                       #T.TunnelAck.IP_Header.HeaderSize := 16#06;
                       #T.TunnelAck.IP_Header.ProtokollVersion := 16#10;
                       #T.TunnelAck.IP_Header.ServiceType := 16#0421;
                       #T.TunnelAck.IP_Header.TotalLaenge := 16#000A;

                       #T.TunnelAck.IP_Body.Laenge := 16#04;
                       #T.TunnelAck.IP_Body.ChannelID := #KNX.ChannelID;
                       #T.TunnelAck.IP_Body.SequenzCount := #KNX.SeqNrEmpf;
                       //#KNX.SeqNr := #T.Tunnel.Conn_Header.SequenzeCount;
                       #T.TunnelAck.IP_Body.Status := 16#0;

                       #POS := 0;
                       #fehler := Serialize(SRC_VARIABLE := #T.TunnelAck, DEST_ARRAY => #SendData, POS := #POS);

                       #SendeLaenge := #POS;
                       #Senden := true;

                   5: //Tunneltelegramm senden!
                       #T.Tunnel.IP_Header.HeaderSize := 16#06;
                       #T.Tunnel.IP_Header.ProtokollVersion := 16#10;
                       #T.Tunnel.IP_Header.ServiceType := 16#420;
                       #T.Tunnel.IP_Header.TotalLaenge := #KNX_Dat.Send_Dat.Laenge+20; //16#15;

                       #T.Tunnel.Conn_Header.Laenge := 04;
                       #T.Tunnel.Conn_Header.ChannelID := #KNX.ChannelID;
                       #T.Tunnel.Conn_Header.SequenzeCount := #KNX.SeqNrSenden;
                       #T.Tunnel.Conn_Header.Reserve := 16#00;

                       #T.Tunnel.Cemi.MessageCode := 16#11;
                       #T.Tunnel.Cemi.AdditionalLaenge := 16#00;
                       #T.Tunnel.Cemi.Kontrollbyte1 := 16#bC;
                       #T.Tunnel.Cemi.Kontrollbyte2 := 16#E0;
                       #T.Tunnel.Cemi.SourceAddr := 16#0000;
                       //#T.Tunnel.Cemi.DestinationAddr := 16#0506;
                       //#T.Tunnel.NPDU.Laenge := 16#01;
                       //#T.Tunnel.NPDU.NPDU_ABCI := 16#00;
                       //IF "Allg".EinAus THEN
                       //    #T.Tunnel.NPDU.Daten[1] := 16#81;
                       //ELSE
                       //    #T.Tunnel.NPDU.Daten[1] := 16#80;
                       //END_IF;

                #T.Tunnel.Cemi.DestinationAddr := #KNX_Dat.Send_Dat.GruppenAddr;
                #T.Tunnel.NPDU.Laenge := #KNX_Dat.Send_Dat.Laenge;
                #T.Tunnel.NPDU.NPDU_ABCI := #KNX_Dat.Send_Dat.NPDU_ABCI;
                #T.Tunnel.NPDU.Daten := #KNX_Dat.Send_Dat.Daten;
                       #POS := 0;
                       #fehler := Serialize(SRC_VARIABLE := #T.Tunnel, DEST_ARRAY => #SendData, POS := #POS);

                       #SendeLaenge := #KNX_Dat.Send_Dat.Laenge+20;
                       #Senden := true;
             6: //Tunnel-Abbau-Telegramm senden
                       #T.AnfTunnelState.IP_Header.HeaderSize := 16#06;
                       #T.AnfTunnelState.IP_Header.ProtokollVersion := 16#10;
                       #T.AnfTunnelState.IP_Header.ServiceType := 16#0209;
                       #T.AnfTunnelState.IP_Header.TotalLaenge := 16#0010;

                       #T.AnfTunnelState.IP_Body.CummunicationChannel := #KNX.ChannelID;
                       #T.AnfTunnelState.IP_Body.Reserve := 16#00;
                       #T.AnfTunnelState.IP_Body.Control_EndPoint.Laenge := 16#08;
                       #T.AnfTunnelState.IP_Body.Control_EndPoint.ProtocolCode := 16#01;
                       #T.AnfTunnelState.IP_Body.Control_EndPoint.IP1 := #EigeneIP[1];
                       #T.AnfTunnelState.IP_Body.Control_EndPoint.IP2 := #EigeneIP[2];
                       #T.AnfTunnelState.IP_Body.Control_EndPoint.IP3 := #EigeneIP[3];
                       #T.AnfTunnelState.IP_Body.Control_EndPoint.IP4 := #EigeneIP[4];
                       #T.AnfTunnelState.IP_Body.Control_EndPoint."Port" := #Port_Lokal;
                       #POS := 0;
                       #fehler := Serialize(SRC_VARIABLE := #T.AnfTunnelState, DEST_ARRAY => #SendData, POS := #POS);

                       #SendeLaenge := #POS;
                       #Senden := true;
           END_CASE;

   //Daten senden!
   #USEND(REQ := #Senden ,
                ID := #ConnID,
                LEN := DINT_TO_UDINT(#SendeLaenge),
                DATA := #SendData,
                ADDR := #KNX_Endpunkt);
   IF #USEND.ERROR THEN
       #Senden := false;
       #STATUS_USEND := #USEND.STATUS;
       #SendeAnf := 0;
   END_IF;
   IF  #USEND.DONE THEN
       #SendeAnf := 0;
       #Senden := false;
       #STATUS_USEND := 0;
       #KNXInfo.SendeTicks := #KNXInfo.SendeTicks + 1;
   END_IF;

   //Bausteinausgaben
   #Status := #State;
   #OK := #State >= 100 AND #State < 250;
   IF #IEC_Timer_TimeOut.Q THEN
       #HMTimeOut := true;
   END_IF;
   IF #URCV.NDR THEN
       #HMTimeOut := false;
   END_IF;
   #TimeOut := #HMTimeOut;
END_FUNCTION_BLOCK

FUNCTION_BLOCK "knx-KO"   // FB15, FBD
{ S7_Optimized_Access := 'TRUE' }
VERSION : 0.1
   VAR_IN_OUT
      Wert : Variant;   // Zu sendender / Empfangender Wert!
      KNX_KO : "KNX_KO";
      KNX_Dat : "KNX_Data_Exchange";
   END_VAR
   VAR
      "knx-SendByChange_Instance" : "knx-SendByChange";
      "knx-rxBus-GroupValueRead_Instance" : "knx-rxBus-GroupValueRead";
      "knx-txBus-GroupValueRead_Instance" : "knx-txBus-GroupValueRead";
      "knx-sendenEmpfangen_Instance" : "knx-sendenEmpfangen";
      fl_counterSend : Bool;
   END_VAR
   VAR_TEMP   // added for the SCL form of the ladder/FBD networks
      _w1 : Bool;
      _w2 : Bool;
   END_VAR
BEGIN

REGION Network 1 (SCL): INFO
   (*

   Sammelbaustein der das KO (Kommunikationsobjekt) zwischen SPS und Bus organisiert


   17.10.2021 van
   Auswertung des #KNX_KO.para.aktiv Bits

   04.10.2021 van
   Baustein erstellt

   *)
END_REGION

REGION Network 2: Aktiv
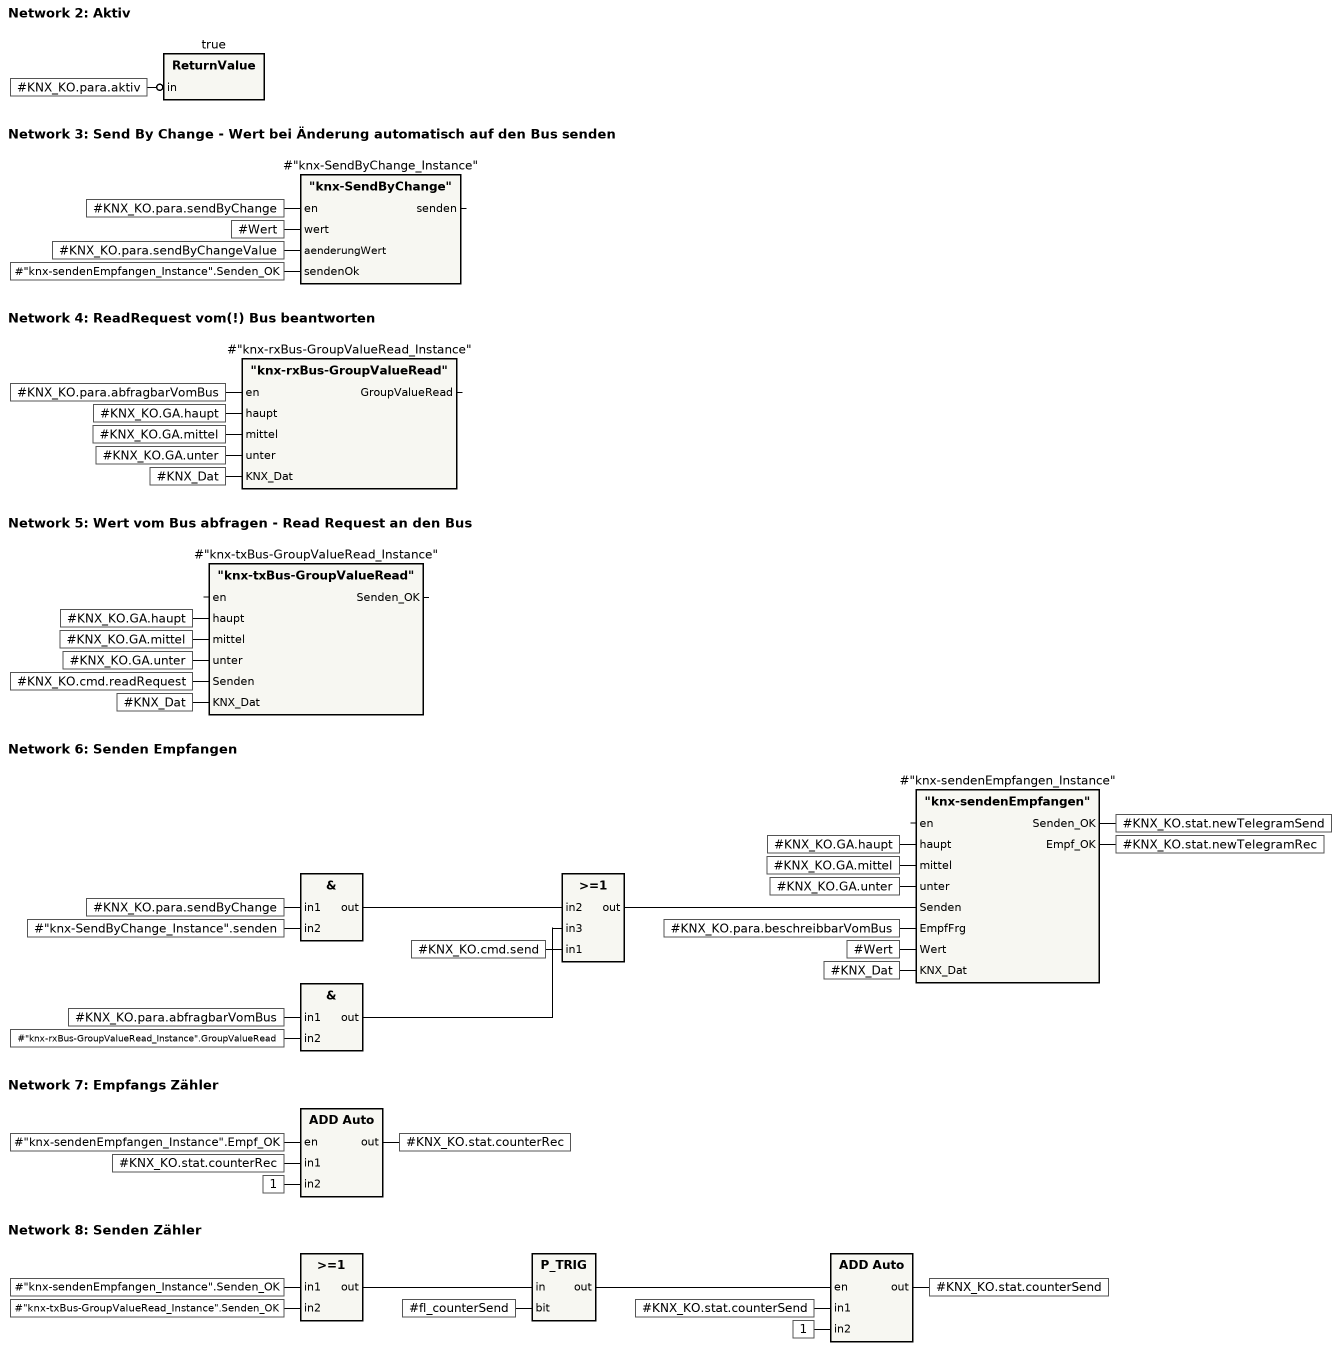
   IF NOT #KNX_KO.para.aktiv THEN
       ENO := true;
       RETURN;
   END_IF;
END_REGION

REGION Network 3: Send By Change - Wert bei Änderung automatisch auf den Bus senden
   IF #KNX_KO.para.sendByChange THEN
       #"knx-SendByChange_Instance"(wert := #Wert,   // "knx-SendByChange"
                               aenderungWert := #KNX_KO.para.sendByChangeValue,
                               sendenOk := #"knx-sendenEmpfangen_Instance".Senden_OK);
   END_IF;
END_REGION

REGION Network 4: ReadRequest vom(!) Bus beantworten
   IF #KNX_KO.para.abfragbarVomBus THEN
       #"knx-rxBus-GroupValueRead_Instance"(haupt := #KNX_KO.GA.haupt,   // "knx-rxBus-GroupValueRead"
                               mittel := #KNX_KO.GA.mittel,
                               unter := #KNX_KO.GA.unter,
                               KNX_Dat := #KNX_Dat);
   END_IF;
END_REGION

REGION Network 5: Wert vom Bus abfragen - Read Request an den Bus
   #"knx-txBus-GroupValueRead_Instance"(haupt := #KNX_KO.GA.haupt,   // "knx-txBus-GroupValueRead"
                           mittel := #KNX_KO.GA.mittel,
                           unter := #KNX_KO.GA.unter,
                           Senden := #KNX_KO.cmd.readRequest,
                           KNX_Dat := #KNX_Dat);
END_REGION

REGION Network 6: Senden Empfangen
   #"knx-sendenEmpfangen_Instance"(haupt := #KNX_KO.GA.haupt,   // "knx-sendenEmpfangen"
                           mittel := #KNX_KO.GA.mittel,
                           unter := #KNX_KO.GA.unter,
                           Senden := (#KNX_KO.para.sendByChange AND #"knx-SendByChange_Instance".senden) OR (#KNX_KO.para.abfragbarVomBus AND #"knx-rxBus-GroupValueRead_Instance".GroupValueRead) OR #KNX_KO.cmd.send,
                           EmpfFrg := #KNX_KO.para.beschreibbarVomBus,
                           Wert := #Wert,
                           KNX_Dat := #KNX_Dat,
                           Senden_OK => #KNX_KO.stat.newTelegramSend,
                           Empf_OK => #KNX_KO.stat.newTelegramRec);
END_REGION

REGION Network 7: Empfangs Zähler
   IF #"knx-sendenEmpfangen_Instance".Empf_OK THEN
       #KNX_KO.stat.counterRec := #KNX_KO.stat.counterRec + 1;
   END_IF;
END_REGION

REGION Network 8: Senden Zähler
   #_w1 := #"knx-sendenEmpfangen_Instance".Senden_OK OR #"knx-txBus-GroupValueRead_Instance".Senden_OK;
   #_w2 := #_w1 AND NOT #fl_counterSend;   // rising edge
   #fl_counterSend := #_w1;
   IF #_w2 THEN #KNX_KO.stat.counterSend := #KNX_KO.stat.counterSend + 1; END_IF;
END_REGION
END_FUNCTION_BLOCK

FUNCTION "knx-GAword-to-GAnr" : "KNX_GA_Nr"   // FC1, SCL
{ S7_Optimized_Access := 'TRUE' }
VERSION : 0.1
   VAR_INPUT
      GruppenAddr : Word;
   END_VAR
BEGIN

   (*

   Wandelt eine Dreistufige KNX GA (Word) in eine ihre Bestandteile (Haupt-, Mittel-, Untergruppe) auf 

   INFOS:

   https://support.knx.org/hc/de/articles/115003188109-Gruppenadressen

   3-Ebenen-Darstellung“ = Hauptgruppe/Mittelgruppe/Untergruppe

   Hauptgruppe = D7+D6+D5+D4+D3 des ersten Oktetts (hohe Adresse)
   Mittelgruppe = D2+D1+D0 des ersten Oktetts (hohe Adresse)
   Untergruppe = das gesamte zweite Oktett (niedrige Adresse)
   Bereiche: Hauptgruppe = 0..31, Mittelgruppe = 0..7, Untergruppe = 0..255

   Quelle:
   https://www.sps-forum.de/gebaeudeautomatisierung/93641-knx-kommunkation-ueber-knxnet-ip-mit-siemens-s7-1500-s7-1200-tia-portal-post704269.html#post704269

   *)



   #"knx-GAword-to-GAnr".haupt := SHR(IN := (#GruppenAddr AND 16#F800), N := 11);
   #"knx-GAword-to-GAnr".mittel := SHR(IN := (#GruppenAddr AND 16#700), N := 8);
   #"knx-GAword-to-GAnr".unter := #GruppenAddr AND 16#FF;
END_FUNCTION

FUNCTION "knx-GAnr-to-GAword" : Word   // FC2, SCL
{ S7_Optimized_Access := 'TRUE' }
VERSION : 0.1
   VAR_INPUT
      haupt : UInt;   // Hauptgruppe = 0..31
      mittel : UInt;   // Mittelgruppe = 0..7
      unter : UInt;   // Untergruppe = 0..255
   END_VAR
   VAR_TEMP
      GruppenAddr : Word;
   END_VAR
BEGIN

   (*

   Erstellt eine Dreistufige KNX GA (Word) aus den Bestandteilen (Haupt-, Mittel-, Untergruppe)

   Quelle:
   Aus "KNX_GruppeAddr" entnommen

   *)


   //Gruppenadresse zu einem Wort zusammenbauen!
   #GruppenAddr := SHL(IN := #haupt, N := 11);
   #GruppenAddr := #GruppenAddr OR SHL(IN := #mittel, N := 8);
   #GruppenAddr := #GruppenAddr OR #unter;


   #"knx-GAnr-to-GAword" := #GruppenAddr;
END_FUNCTION

FUNCTION "knx-real-to-DPT9" : Word   // FC3, SCL
{ S7_Optimized_Access := 'TRUE' }
VERSION : 0.1
   VAR_INPUT
      inReal : Real;
   END_VAR
   VAR_TEMP
      tmpExp : Int;
      tmpDIntValIn : DInt;
      tmp_dInt : DInt;
      tmpOut : Int;
   END_VAR
BEGIN

   (*

   Wandelt eine Real Zahl in den DPT9.xxx (2 Byte Gleitkommawert)

   Quelle:
   https://www.sps-forum.de/threads/knx-kommunkation-%C3%BCber-knxnet-ip-mit-siemens-s7-1500-s7-1200-tia-portal.93641/post-804342

   Weitere Infos:
   03_07_02 Datapoint Types v01.08.02 AS.pdf
   3.10 Datapoint Types “2-Octet Float Value”

   Range: [-671 088,64 … 670 760,96]


   03.10.2021 van
   Baustein erstellt anhand des Code von Oberchefe

   *)

   #tmpExp := 0;    (*    Exponent initialisieren    *)

   #tmpDIntValIn := REAL_TO_DINT(#inReal * 100.0);

   IF #tmpDIntValIn > 2047  THEN   // OR #tmpDIntValIn < -2048

       WHILE #tmpDIntValIn / (2**#tmpExp) > 2047 DO     //EXPT(2, #tmpExp)
           #tmpExp := #tmpExp + 1;
       END_WHILE;

   ELSIF #tmpDIntValIn < -2048 THEN

       WHILE #tmpDIntValIn / (2**#tmpExp) < -2048 DO    // EXPT(2, #tmpExp)
           #tmpExp := #tmpExp + 1;
       END_WHILE;

   ELSE            (*    Kein Exponent erforderlich    *)

       ;

   END_IF;


   #tmp_dInt := #tmpDIntValIn / REAL_TO_DINT((2**(#tmpExp)));         (*    Mantisse roh   *)  //(EXPT(2, INT_TO_WORD(#tmpExp))

   #tmp_dInt := WORD_TO_DINT(DINT_TO_WORD(#tmp_dInt) AND 16#7FF);
   #tmpOut := SHL(IN := #tmpExp, N:=11);                (*    Exponent positionieren        *)


   IF #tmpDIntValIn < 0 THEN                    (*    negativ?    -> Vorzeichen setzen    *)
       #tmpOut := #tmpOut OR 16#8000;
   END_IF;


   #"knx-real-to-DPT9":= #tmpOut OR DINT_TO_WORD(#tmp_dInt);
END_FUNCTION

FUNCTION "knx-DPT9-to-real" : Real   // FC4, SCL
{ S7_Optimized_Access := 'TRUE' }
VERSION : 0.1
   VAR_INPUT
      inWord : Word;
   END_VAR
   VAR_TEMP
      tmp_Word1 : Word;
      tmp_M : DWord;
      tmp_Dword : DWord;
      tmp_e2 : UDInt;
      tmp_Real : Real;
      tmp_Int : Int;
      tmpInt_M : Int;
      tmpInt_E : Int;
      tmpReal_M : Real;
      tmpReal_E : Real;
      tmpReal : Real;
   END_VAR
BEGIN
   (*

   Wandelt ein DPT9.xxx (2 Byte Gleitkommawert) in einen Real

   Weitere Infos:
   03_07_02 Datapoint Types v01.08.02 AS.pdf
   3.10 Datapoint Types “2-Octet Float Value”

   03.10.2021 van
   Baustein erstellt

   *)



   //Ergebnis = (0,01 * M)*2^E   //Siehe PDF 03_07_02 Kap. 3.10)
   // E = [0 … 15]
   // M = [-2 048 … 2 047], two’s complement notation

   (*

   76543210 76543210
   MEEEEMMM MMMMMMMM

   *)

   #tmp_Word1:= #inWord;

   // Mantisse
   #tmpInt_M := WORD_TO_INT(#tmp_Word1 & 16#07ff);
   #tmpReal_M := INT_TO_REAL(#tmpInt_M);

   //Negative Mantisse anpassen
   //Das muss noch irgendwie besser gehen ...
   IF #tmp_Word1.%X15 THEN
       #tmpReal_M := (#tmpReal_M*-1.0) + 2048.0;
   END_IF;


   // Exponent
   // #tmp_Dword := #tmp_Word1 & 16#7800;  //Exponent
   // #tmp_e2 := SHR(IN := #tmp_Dword, N := 11);

   #tmp_e2 := SHR(IN := SHL(IN := #tmp_Word1, N := 1), N := 12);

   #tmpInt_E := UDINT_TO_INT(#tmp_e2);
   #tmpReal_E := INT_TO_REAL(#tmpInt_E);


   // FloatValue = (0,01 * M)*2^E 
   #tmpReal := (0.01 * #tmpReal_M) * (2**#tmpReal_E);


   //Vorzeichen
   IF #tmp_Word1.%X15 THEN
       #tmpReal := (#tmpReal * -1.0) ;
   END_IF;


   #"knx-DPT9-to-real" := #tmpReal;
END_FUNCTION

FUNCTION "knx-DPT3-to-plc" : "KNX_DPT3"   // FC14, SCL
{ S7_Optimized_Access := 'TRUE' }
VERSION : 0.1
   VAR_INPUT
      data : Byte;   // RAW DPT3 Daten
   END_VAR
   VAR_TEMP
      tmpStepCode : USInt;
   END_VAR
   // Ret_Val : Aufbereitete DPT3 Daten
BEGIN
   (*

   knx-DPT3-to-plc

   Wandelt den DPT3 Wert vom KNX Bus in einen PLC "KNX_DPT3" Wert

   DPT 3   4 Bit   0..15     
   3.yyy = boolesch + vorzeichenloser 3-Bit-Wert, z. B. Auf-/Abdimmen  

   \The KNX Standard v2.1\The KNX Standard v2.1\03 Volume 3 System Specifications\
   03_07_02 Datapoint Types v01.08.02 AS.pdf
   3.3 Datapoint Types B1U3 


   20.02.2024 van
   Baustein erstellt

   *)

   (*** StepCode ***

   StepCode The amount of intervals into which the 
   range of 0 % … 100 % is subdivided, or the 
   break indication. 

   - 001b…111b: Step Number of intervals = 2^(stepcode-1) 
   - 000b: Break 

   *)


   // Daten aufbereiten
   #tmpStepCode.%X0 := #data.%X0;
   #tmpStepCode.%X1 := #data.%X1;
   #tmpStepCode.%X2 := #data.%X2;

   #"knx-DPT3-to-plc".prozent:= FLOOR(100.0 / (2**(#tmpStepCode-1)));


   (*** c ***

   3.007 DPT_Control_Dimming 
   c Increase or decrease the brightness. 
   0 = Decrease 
   1 = Increase 

   3.008 DPT_Control_Blinds 
   c Move up or down. 
   0 = Up 
   1 = Down 

   *)

   // Daten aufbereiten
   #"knx-DPT3-to-plc".Down_Increase := #data.%X3;
END_FUNCTION

FUNCTION "knx-plc-to-DPT3" : Byte   // FC15, SCL
{ S7_Optimized_Access := 'TRUE' }
VERSION : 0.1
   VAR_INPUT
      data : "KNX_DPT3";   // Aufbereitete DPT3 Daten
   END_VAR
   VAR_TEMP
      tmpStepCode : USInt;
   END_VAR
   // Ret_Val : RAW DPT3 Daten
BEGIN
   (*

   knx-plc-to-DPT3

   Wandelt einen PLC "KNX_DPT3" Wert in einen KNX Bus DPT3 Wert 


   DPT 3   4 Bit   0..15     
   3.yyy = boolesch + vorzeichenloser 3-Bit-Wert, z. B. Auf-/Abdimmen  

   \The KNX Standard v2.1\The KNX Standard v2.1\03 Volume 3 System Specifications\
   03_07_02 Datapoint Types v01.08.02 AS.pdf
   3.3 Datapoint Types B1U3 


   21.02.2024 van
   Baustein erstellt

   *)

   (*** StepCode ***

   StepCode The amount of intervals into which the 
   range of 0 % … 100 % is subdivided, or the 
   break indication. 

   - 001b…111b: Step Number of intervals = 2^(stepcode-1) 
   - 000b: Break 

   *)


   // Daten aufbereiten

   // 1, 3, 6, 12, 25, 50, 100% / 0 = Stopp

   CASE #data.prozent OF
       1..2:  // 
           #tmpStepCode := 7;
       3..5:  // 
           #tmpStepCode := 6;
       6..11:  // 
           #tmpStepCode := 5;
       12..24:  // 
           #tmpStepCode := 4;
       25..49:  // 
           #tmpStepCode := 3;
       50..99:  // 
           #tmpStepCode := 2;
       100:  // 
           #tmpStepCode := 1;
       ELSE  // 
           #tmpStepCode := 0;
   END_CASE;


   #"knx-plc-to-DPT3".%X0 := #tmpStepCode.%X0;
   #"knx-plc-to-DPT3".%X1 := #tmpStepCode.%X1;
   #"knx-plc-to-DPT3".%X2 := #tmpStepCode.%X2;



   (*** c ***

   3.007 DPT_Control_Dimming 
   c Increase or decrease the brightness. 
   0 = Decrease 
   1 = Increase 

   3.008 DPT_Control_Blinds 
   c Move up or down. 
   0 = Up 
   1 = Down 

   *)

   // Daten aufbereiten
   #"knx-plc-to-DPT3".%X3 := #data.Down_Increase;
END_FUNCTION